{attribute addProperty BoxType "EL2602-0000-0016"}
{attribute addProperty Id "ChannelAT %Q*ARRAY[0..1] OF Channel_7F374EB01620WcStateAT %I*WcState_28A8677510.1250InfoDataAT %I*InfoData_192954DE1620"}
{attribute addProperty CRC "2824189094"}
{attribute addProperty SizeInBites "33"}
{attribute addProperty SizeInBytes "4.125"}
TYPE EL2602_39EC201D :
STRUCT
	{attribute addProperty Name "Channel"}
	Channel : ARRAY[0..1] OF Channel_7F374EB0;
	{attribute addProperty Name "WcState"}
	WcState : WcState_28A86775;
	{attribute addProperty Name "InfoData"}
	InfoData : InfoData_192954DE;
END_STRUCT
END_TYPE

(* stored: Version 1.2.0.0, ProductVersion 3.1.4024.9
   DUT EL2602_39EC201D: Id {c0b22098-6b01-461a-b917-a4d78a0a57d6} *)
